FUNCTION_BLOCK PUBLIC FB_LampSetDirectDALI EXTENDS FB_LampSetDirect
VAR
END_VAR

// Sets the control value of the DALI lamp to a value between 0 and 254.
METHOD PUBLIC SetLightLevel
VAR_INPUT
	nNewLightLevel		: BYTE(0..254);
END_VAR
nLightLevel := nNewLightLevel;
END_METHOD

END_FUNCTION_BLOCK

(* stored: Version 1.1.0.1, ProductVersion 3.1.4024.11
   POU FB_LampSetDirectDALI: Id {508b93c0-0778-4ff1-aedf-858d8647b6a3}, SpecialFunc None
   Method SetLightLevel: Id {fcb47fde-6ee2-43a2-b668-4bd49ce3e7e1} *)
